FUNCTION MatTranspose : Mat3
VAR_INPUT
	m : Mat3;
END_VAR
VAR
	i, j : INT;
END_VAR

FOR i := 0 TO 2 DO
	FOR j := 0 TO 2 DO
		MatTranspose.data[j, i] := m.data[i, j];
	END_FOR
END_FOR

END_FUNCTION

(* stored: Version 1.1.0.1, ProductVersion 3.1.4024.2
   POU MatTranspose: Id {e8b3e56d-ffa0-4e92-9e7e-d00c9b8c618d}, SpecialFunc None *)
